// TwinCAT 3 PLC project Serie_3
// ProgramVersion: 3.1.4022.3
// libraries:
//   Tc2_Standard, * (Beckhoff Automation GmbH)
//   Tc2_System, * (Beckhoff Automation GmbH)
//   Tc3_Module, * (Beckhoff Automation GmbH)
// project tree:
//   DUTs/ SafeState.TcDUT
//   GVLs/ GVL.TcGVL
//   / PlcTask.TcTTO
//   POUs/ AdditionFunction.TcPOU, EdgeDetector.TcPOU, MAIN.TcPOU
//   POUs/POUs/ EdgeDetector_1.TcPOU
// real-time tasks:
//   TASK PlcTask: cycle T#10ms, priority 20, ADS port 350
// I/O:
//   DEVICE Gerät 1 (EtherCAT), AmsNetId 5.12.140.184.2.1
//     Klemme 1 (EK1200) [EK1200-5000 EtherCAT Netzteil (2A E-Bus)]
//       Klemme 2 (EL1004) [EL1004 4K. Dig. Eingang 24V, 3ms]
//       Klemme 3 (EL2004) [EL2004 4K. Dig. Ausgang 24V, 0.5A]
//       Klemme 4 (EL3004) [EL3004 4K.Ana. Eingang  +/-10V]
//       Klemme 5 (EL4034) [EL4034 4K. Ana. Ausgang +/-10V, 12bit]
//       Klemme 6 (EK1110) [EK1110 EtherCAT-Verlängerung]
// variable links:
//   Serie_3/Serie_3 Instance <-> Device 1 (EtherCAT)/Term 1 (EK1200)/Term 2 (EL1004)
//     PlcTask Inputs/GVL.b_buttonBlue <-> Channel 2/BlueButton
//     PlcTask Inputs/GVL.b_buttonYellow <-> Channel 1/YellowButton
//   Serie_3/Serie_3 Instance <-> Device 1 (EtherCAT)/Term 1 (EK1200)/Term 3 (EL2004)
//     PlcTask Outputs/GVL.b_LampeCorrect <-> Channel 2/GreenLight
//     PlcTask Outputs/GVL.b_LampeWrong <-> Channel 1/RedLight

CONFIGURATION Serie_3
    RESOURCE PLC ON TwinCAT3
        TASK PlcTask(INTERVAL := T#10ms, PRIORITY := 20);
        PROGRAM MAIN WITH PlcTask : MAIN;
    END_RESOURCE
END_CONFIGURATION

// ---- DUTs/SafeState.TcDUT
{attribute 'qualified_only'}
{attribute 'strict'}
TYPE SafeState :
(
	Init := 0,
	Close := 1,
	Open := 2,
	CheCkDigit := 3,
	WrongCode := 4
);
END_TYPE

// ---- GVLs/GVL.TcGVL
{attribute 'qualified_only'}
VAR_GLOBAL
	b_buttonYellow AT %I* : BOOL;
	b_buttonBlue AT %I* : BOOL;
	b_LampeCorrect AT %Q* : BOOL;
	b_LampeWrong AT %Q* : BOOL;
	bA_CodePins : ARRAY [1..4] OF BOOL;
	i_currentIndex : INT;
	i_correctCounter : INT;
	i_lightDuration : INT := 5000;		// ms
END_VAR

// ---- POUs/MAIN.TcPOU
PROGRAM MAIN
VAR
	b_YelloPushed : BOOL;
	b_BluePushed : BOOL;
	byte_decider : BYTE;
	i_EdgdetectorYellow : EdgeDetector_1;
	i_EdgdetectorBlue : EdgeDetector_1;
	b_risingEdge : BOOL;
	state : SafeState;
END_VAR

i_EdgdetectorYellow();
i_EdgdetectorYellow.inputValue := GVL.b_buttonYellow;
b_YelloPushed := i_EdgdetectorYellow.riesingEdge;
i_EdgdetectorBlue();
i_EdgdetectorBlue.inputValue := GVL.b_buttonBlue;
b_BluePushed := i_EdgdetectorBlue.riesingEdge;
IF b_YelloPushed OR b_BluePushed THEN
	b_risingEdge := TRUE;
	ELSE
	b_risingEdge := FALSE;
END_IF
CASE state OF
	0 : GVL.bA_CodePins[1] := TRUE;		// State = Init
		GVL.bA_CodePins[2] := FALSE;
		GVL.bA_CodePins[3] := FALSE;
		GVL.bA_CodePins[4] := TRUE;
		state :=1 ;		
	1 : GVL.b_LampeCorrect := FALSE;	// State = Close
		GVL.b_LampeWrong := FALSE;
		GVL.i_correctCounter := 0;
		GVL.i_currentIndex := 1;
		GVL.i_lightDuration := 5000;
		state :=3;		
	2 : IF GVL.i_lightDuration >0 THEN						// State = CorrectCode
		GVL.b_LampeCorrect := TRUE;							// Turn the Green 	
		GVL.i_lightDuration := GVL.i_lightDuration -10;
		ELSE
		GVL.b_LampeCorrect := FALSE;
		state :=1;				// Time is Over > Next state > Close		
		END_IF
	3 : IF b_risingEdge THEN	// State = CheCkDigit
		CASE GVL.i_currentIndex OF
			1 : IF GVL.bA_CodePins[GVL.i_currentIndex] = b_YelloPushed THEN
				GVL.i_currentIndex := GVL.i_currentIndex +1;
				ELSE
					state := 4;	
				END_IF
			2 : IF GVL.bA_CodePins[GVL.i_currentIndex] = NOT b_BluePushed THEN
				GVL.i_currentIndex := GVL.i_currentIndex +1;
				ELSE
					state := 4;	
				END_IF
			3 : IF GVL.bA_CodePins[GVL.i_currentIndex] = NOT b_BluePushed THEN
				GVL.i_currentIndex := GVL.i_currentIndex +1;
				ELSE
					state := 4;	
				END_IF
			4 : IF GVL.bA_CodePins[GVL.i_currentIndex] = b_YelloPushed THEN
					state := 2;	
				ELSE
					state := 4;	
				END_IF		
		END_CASE
		ELSE
		state := 3;		// no button detected > dont change State.
		END_IF
	4 : IF GVL.i_lightDuration >0 THEN						// State = WrongCode
		GVL.b_LampeWrong := TRUE;							// Turn the Red 	
		GVL.i_lightDuration := GVL.i_lightDuration -10;
		ELSE
		GVL.b_LampeWrong := FALSE;
		state :=1;				// Time is Over > Next state > Close		
		END_IF
END_CASE

END_PROGRAM

// ---- POUs/POUs/EdgeDetector_1.TcPOU
FUNCTION_BLOCK EdgeDetector_1
VAR_INPUT
	inputValue : BOOL ;
END_VAR

VAR_OUTPUT
	riesingEdge :BOOL;
	fallingEdge :BOOL;
END_VAR
VAR
	safeStatus:BOOL;
	totzeit : INT;
END_VAR

fallingEdge := FALSE;
riesingEdge := FALSE;
IF totzeit <1 THEN
	IF safeStatus = FALSE AND inputValue = TRUE THEN
		riesingEdge:= TRUE;
		totzeit := 100;
	ELSIF safeStatus = TRUE AND inputValue = FALSE THEN
		fallingEdge:= TRUE;
		totzeit := 100;
	END_IF
	ELSE
	totzeit := totzeit -1;
END_IF
safeStatus := inputValue;

END_FUNCTION_BLOCK

// ---- POUs/AdditionFunction.TcPOU
FUNCTION AdditionFunction : REAL
VAR_INPUT
	i_rValueA : REAL;
	i_rValueB : REAL;
END_VAR
VAR
END_VAR

AdditionFunction := i_rValueA + i_rValueB;

END_FUNCTION

// ---- POUs/EdgeDetector.TcPOU
FUNCTION_BLOCK EdgeDetector
VAR_INPUT
	b_StateButtonActal : BOOL;
END_VAR
VAR_OUTPUT
	s_StateEdgedetector: STRING;
END_VAR
VAR
	b_StateButtonOld : BOOL;
END_VAR

IF NOT b_StateButtonOld AND b_StateButtonActal THEN
	s_StateEdgedetector := 'risingEdge';
	
ELSIF  b_StateButtonOld AND NOT b_StateButtonActal THEN
	s_StateEdgedetector := 'falingEdge';
ELSE 
	s_StateEdgedetector := 'not Changed';
END_IF
b_StateButtonOld := b_StateButtonActal;

END_FUNCTION_BLOCK
